VAR_GLOBAL
	Trace : Trace<ApplicationBaseParameter.MaxCountInCollections> := (TraceLevel := ApplicationBaseParameter.TraceLevel);
	{attribute 'hide'}
	TcEventLogger : TcEventLogger(Trace);
	{attribute 'hide'}
	AdsLogger : AdsLogger(Trace);
END_VAR

(* stored: Version 1.1.0.1, ProductVersion 3.1.4026.18
   GVL CoreTrace: Id {a08d82f5-c40f-43ad-8071-187f0f8bb6e7} *)
